(* CODESYS project EcoWatt.library
   Description: This library retrieve EcoWatt indicators from RTE.
   Author: quenorha
   Version: 1.0.0.0
   Company: WAGO_FR
   Title: EcoWatt
   Placeholder: EcoWatt
   DocFormat: reStructuredText
   DefaultNamespace: EcoWatt

Project tree, tasks and I/O mapping:
  libraries: WagoSysVersion, 1.0.0.0 (WAGO); WagoAppJSON, 1.1.0.25 (WAGO); WagoAppString, 1.6.3.4 (WAGO); WagoAppTime, 1.7.3.5 (WAGO); WagoAppHTTP, 1.7.3.4 (WAGO)
  10 Documentation/
    function block Help [ST]
  20 Program Organization Units/
    function block FbEcoWatt [ST]
  80 Data Types/
    data type typDayEcoWatt
  30 Visualizations/
    visualisation EcoWattDay
    visualisation EcoWattHour
    visualisation EcoWattVisu
  90 Internal/
    function block FbEcoWattJSON_Handler [ST]: JSON_KeyDetected, JSON_ValueDetected
    function FuCustomFormatToDT [ST]
    function FuDTToCustomFormat [ST]
  global variables VersionHistory
  Images/
    WAGO
  00000000-0000-0000-0000-000000000000|C:\Users\u044132\Downloads\old PC\Pictures\WAGO.bmp
  text list GlobalTextList
*)

// 80 Data Types/typDayEcoWatt
TYPE typDayEcoWatt :
STRUCT
		sMessage : STRING(1024);
		dtGenDate : DT;
		dtForecastDay : DT;
		bDayValue :BYTE;
		abForecast : ARRAY [0..23] OF BYTE; 
END_STRUCT
END_TYPE

// VersionHistory
(* 

**EcoWatt.library**

Description: Library for  WAGO I/O- System 

============ =========== ====================== =================
**date**     **version** **author**             **change**       
------------ ----------- ---------------------- -----------------
11.10.2022	   1.0.0.0       quenorha          First version
============ =========== ====================== =================

**Known Bugs**
   - 
   - 

**To-Do's**
   - 
   - 

*)

VAR_GLOBAL
	Info : ProjectInfo('1.0.0.0','EcoWatt.library',sLicense:='WAGO');
END_VAR

(*

11.10.2022	   1.0.0.0       quenorha          
	* [NEW] First version
	* [FIXED] ....

*)

// 90 Internal/FbEcoWattJSON_Handler
(*
	This function block uses the methods JSON_Key_Detected, JSON_ObjcectClosed and JSON_ValueDetected to import the values of
	interest to the appropriate function block.

	
*)
FUNCTION_BLOCK FbEcoWattJSON_Handler EXTENDS FbJSON_Handler
VAR_IN_OUT
	atypEcoWatt : ARRAY [0..3] OF typDayEcoWatt;
END_VAR
VAR
	parserState					: INT;	
	m							: INT;
	bDay : INT;
	bHour: INT;
END_VAR

(*

**Function**

	
**Graphical Illustration**

	.. wago.autoimage::
	
*)
METHOD JSON_KeyDetected 
VAR_INPUT
	sJSON_Object			:	STRING; // JSON object detected
END_VAR

VAR

END_VAR


IF sJSON_Object='signals' THEN	
	parserstate:=0;// jetzt kommt der Wert
ELSIF sJSON_Object='GenerationFichier' THEN	
	parserstate:=1;// jetzt kommt der Wert
ELSIF sJSON_Object='jour' THEN	
	parserstate:=2;// jetzt kommt der Wert
ELSIF sJSON_Object='dvalue' THEN	
	parserstate:=3;// jetzt kommt der Wert	
ELSIF sJSON_Object='message' THEN	
	parserstate:=4;// jetzt kommt der Wert
ELSIF sJSON_Object='values' THEN	
	parserstate:=5;// jetzt kommt der Wert
ELSIF sJSON_Object='pas' THEN	
	parserstate:=6;// jetzt kommt der Wert	
ELSIF sJSON_Object='hvalue' THEN	
	parserstate:=7;// jetzt kommt der Wert
END_IF
END_METHOD

(*

**Function**

	

**Graphical Illustration**

	.. wago.autoimage::
	
*)
METHOD JSON_ValueDetected 
VAR_INPUT
	sJSON_Value			:	STRING(JSON_MAX_STRING_SAX); // JSON value detected
END_VAR

VAR

END_VAR
{warning disable C0371}
IF __ISVALIDREF(atypEcoWatt)=FALSE THEN
	RETURN;
END_IF

CASE parserState OF
	0: bDay:=0 ;
	   bHour:=0;
	
	1:atypEcoWatt[bDay].dtGenDate:=FuCustomFormatToDT(sDateTimeString:=sJSON_Value,sCustomFormat:='AAAA-MM-JJThh:mm:SS');
	
	2:atypEcoWatt[bDay].dtForecastDay:=FuCustomFormatToDT(sDateTimeString:=sJSON_Value,sCustomFormat:='AAAA-MM-JJThh:mm:SS');
		
	3:atypEcoWatt[bDay].bDayValue:=TO_BYTE(sJSON_Value);
	
	4:atypEcoWatt[bDay].sMessage:=sJSON_Value;
		
	5://atypEcoWatt[bDay].abForecast[bHour]:=TO_BYTE(sJSON_Value);
		
	
	6:bHour:=TO_BYTE(sJSON_Value);
		
	7:atypEcoWatt[bDay].abForecast[bHour]:=TO_BYTE(sJSON_Value);
		IF bHour=23 THEN
			bDay:=bDay+1;
		END_IF

END_CASE
{warning enable C0371}
END_METHOD

END_FUNCTION_BLOCK

// 90 Internal/FuCustomFormatToDT
FUNCTION FuCustomFormatToDT : DT
(*This function returns the date/time value into a string formated with a customizable format, for example JJ/MM/AA,HH:mm:SS*)
VAR_INPUT
	sDateTimeString :  STRING ; (*Date/Time to format*)
	sCustomFormat : STRING :='JJ/MM/AA,HH:mm:SS'; (*Date/Time format to use, for example JJ/MM/AA,HH:mm:SS*)
END_VAR
VAR
	sYear : STRING(4);
	sShortYear : STRING(2);
 	sMonth :  STRING(2);
	sDay : STRING(2);
	sHour : STRING(2);
	sMinute : STRING(2);
	sSecond : STRING(2);
	sTemp:STRING;
	sTempResult : STRING;
	sSeparator : STRING(1);
	sFormat : STRING;
	i : INT;
	xAdd : BOOL;
	
	iPos : INT;
	iLength : INT;
	bSecond: BYTE;
	bMinute: BYTE;
	bHour: BYTE;
	bMonth: BYTE;
	bDay: BYTE;
	wYear: WORD;
END_VAR

IF sDateTimeString='' THEN
	FuCustomFormatToDT:=dt#1970-01-01-00:00:00;
ELSE
	iPos:=FIND(sCustomFormat,'SS');
	IF iPos=0 THEN
		iPos:=FIND(sCustomFormat,'ss');	
	END_IF
	IF iPos=0 THEN
		sSecond:='00';
	ELSE
		sSecond:=MID(sDateTimeString,2,iPos);
	END_IF
	bSecond:=STRING_TO_BYTE(sSecond);
		
	iPos:=FIND(sCustomFormat,'mm');
	IF iPos=0 THEN
		sMinute:='00';
	ELSE
		sMinute:=MID(sDateTimeString,2,iPos);
	END_IF
	bMinute:=STRING_TO_BYTE(sMinute);
		
	iPos:=FIND(sCustomFormat,'HH');
	IF iPos=0 THEN
		iPos:=FIND(sCustomFormat,'hh');	
	END_IF
	IF iPos=0 THEN
		sHour:='00';
	ELSE
		sHour:=MID(sDateTimeString,2,iPos);
	END_IF
	bHour:=STRING_TO_BYTE(sHour);
	
	
	iPos:=FIND(sCustomFormat,'MM');
	IF iPos=0 THEN
		sMonth:='00';
	ELSE
		sMonth:=MID(sDateTimeString,2,iPos);
	END_IF
	bMonth:=STRING_TO_BYTE(sMonth);
		
	iPos:=FIND(sCustomFormat,'JJ');
	IF iPos=0 THEN
		iPos:=FIND(sCustomFormat,'jj');	
	END_IF
	IF iPos=0 THEN
		sDay:='00';
	ELSE
		sDay:=MID(sDateTimeString,2,iPos);
	END_IF
	bDay:=STRING_TO_BYTE(sDay);	
	
	iPos:=FIND(sCustomFormat,'AAAA');
	iLength:=4;
	IF iPos=0 THEN
		iPos:=FIND(sCustomFormat,'aaaa');
		iLength:=4;	
	END_IF
	IF iPos=0 THEN
		iPos:=FIND(sCustomFormat,'AA');
		iLength:=2;	
	END_IF
	IF iPos=0 THEN
		iPos:=FIND(sDateTimeString,'aa');
		iLength:=2;	
	END_IF
	IF iPos=0 THEN
		sYear:='00';
	ELSE
		sYear:=MID(sDateTimeString,iLength,iPos);
	END_IF
	IF iLength=2 THEN
		wYear:=STRING_TO_WORD(sYear);
		wYear:=wYear+2000;		
	ELSE	
		wYear:=STRING_TO_WORD(sYear);	
	END_IF
	
	FuCustomFormatToDT:=FuFormatToDT(bDay,bMonth,TO_INT(wYear),bHour,bMinute,bSecond);	
END_IF

END_FUNCTION

// 10 Documentation/Help
(*

.. note::  Note

**Bibliothèque EcoWatt**
///Cette bibliothèque permet de Récupérer les informations du signal EcoWatt fournies par RTE. 
///Créer un compte sur https://data.rte-france.com/catalog/-/api/consumption/Ecowatt/v4.0
///S'abonner à l'API EcoWatt. 
///Dans "mes applications", Cliquer sur Copier en base 64 pour récupérer l'identifiant. 
///Le renseigner au niveau de sBase64Code.
///Lorsque xUpdate est activé, la requête de récupération du jeton est effectué, puis la requête de récupération des données. 
///xUpdate retombe à FALSE lorsque la requête est effectuée ou si il y a une erreur.

///Les valeurs numériques retournées correspondent aux niveaux suivant : 
/// - 1) Vert : La consommation est normale
/// - 2) Orange : le système électrique est tendu : "écogestes" bienvenus.
/// - 3) Rouge : le système électrique est très tendu, coupures inévitables si la consommation n'est pas réduite. 
///bCurrentEcoWattValue et bextEcoWattValue fournissent la valeur EcoWatt de l'heure en cours et de l'heure suivante. 
///Attention à faire en sorte de rafraichir les données périodiquement en activant xUpdate. 
///L'API ne peut être appelée que toutes les 15 minutes. Au delà de ce quota, le code HTTP 429 sera renvoyé.

	
.. figure:: ../../images/WAGO.bmp
	:align: center
	:alt: descriptif de l'image
	
*)
FUNCTION_BLOCK Help

END_FUNCTION_BLOCK

// 20 Program Organization Units/FbEcoWatt

///Cette bibliothèque permet de Récupérer les informations du signal EcoWatt fournies par RTE. 
///Créer un compte sur https://data.rte-france.com/catalog/-/api/consumption/Ecowatt/v4.0
///S'abonner à l'API EcoWatt. 
///Dans "mes applications", Cliquer sur Copier en base 64 pour récupérer l'identifiant. 
///Le renseigner au niveau de sBase64Code.
///Lorsque xUpdate est activé, la requête de récupération du jeton est effectué, puis la requête de récupération des données. 
///xUpdate retombe à FALSE lorsque la requête est effectuée ou si il y a une erreur.

///Les valeurs numériques retournées correspondent aux niveaux suivant : 
/// - 1) Vert : La consommation est normale
/// - 2) Orange : le système électrique est tendu : "écogestes" bienvenus.
/// - 3) Rouge : le système électrique est très tendu, coupures inévitables si la consommation n'est pas réduite. 
///bCurrentEcoWattValue et bextEcoWattValue fournissent la valeur EcoWatt de l'heure en cours et de l'heure suivante. 
///Attention à faire en sorte de rafraichir les données périodiquement en activant xUpdate. 
///L'API ne peut être appelée que toutes les 15 minutes. Au delà de ce quota, le code HTTP 429 sera renvoyé.

FUNCTION_BLOCK FbEcoWatt
VAR_INPUT
	sBase64Code : STRING(255); //Identifiant API RTE au format base 64.
END_VAR
VAR_IN_OUT 
	xUpdate: BOOL;				// Rafraichit les données - retombe automatiquement. 
END_VAR
VAR_OUTPUT
	atypEcoWatt : ARRAY [0..3] OF typDayEcoWatt; // Données EcoWatt aujourd'hui, et jusqu'à J+3
	bCurrentEcoWattValue : BYTE;   // Indicateur EcoWatt heure en cours 
	bNextEcoWattValue : BYTE; // Indicateur EcoWatt heure suivante
	xError : BOOL;
	sErrorDesc: STRING;
END_VAR
VAR
	oFbHTTPs_Get_Token: WagoAppHTTP.FbHTTPs_Get;
	xTriggerToken: BOOL;
	sBuffer : STRING(3000);
	sExempleData : STRING(3000):='{"signals": [{"GenerationFichier": "2022-10-10T07:36:25+02:00","jour": "2022-10-10T00:00:00+02:00","dvalue": 1,"message": "Situation normale ","values": [{"pas": 0,"hvalue": 1},{"pas": 1,"hvalue": 1},{"pas": 2,"hvalue": 1},{"pas": 3,"hvalue": 1},{"pas": 4,"hvalue": 1},{"pas": 5,"hvalue": 1},{"pas": 6,"hvalue": 1},{"pas": 7,"hvalue": 1},{"pas": 8,"hvalue": 1},{"pas": 9,"hvalue": 1},{"pas": 10,"hvalue": 1},{"pas": 11,"hvalue": 1},{"pas": 12,"hvalue": 1},{"pas": 13,"hvalue": 1},{"pas": 14,"hvalue": 1},{"pas": 15,"hvalue": 1},{"pas": 16,"hvalue": 1},{"pas": 17,"hvalue": 1},{"pas": 18,"hvalue": 1},{"pas": 19,"hvalue": 1},{"pas": 20,"hvalue": 1},{"pas": 21,"hvalue": 1},{"pas": 22,"hvalue": 1},{"pas": 23,"hvalue": 1}]},{"GenerationFichier": "2022-10-11T07:36:25+02:00","jour": "2022-10-11T00:00:00+02:00","dvalue": 3,"message": "Coupures d$'électricité programmées","values": [{"pas": 0,"hvalue": 1},{"pas": 1,"hvalue": 1},{"pas": 2,"hvalue": 1},{"pas": 3,"hvalue": 1},{"pas": 4,"hvalue": 1},{"pas": 5,"hvalue": 2},{"pas": 6,"hvalue": 2},{"pas": 7,"hvalue": 3},{"pas": 8,"hvalue": 3},{"pas": 9,"hvalue": 3},{"pas": 10,"hvalue": 3},{"pas": 11,"hvalue": 3},{"pas": 12,"hvalue": 3},{"pas": 13,"hvalue": 2},{"pas": 14,"hvalue": 2},{"pas": 15,"hvalue": 2},{"pas": 16,"hvalue": 2},{"pas": 17,"hvalue": 3},{"pas": 18,"hvalue": 3},{"pas": 19,"hvalue": 3},{"pas": 20,"hvalue": 2},{"pas": 21,"hvalue": 2},{"pas": 22,"hvalue": 2},{"pas": 23,"hvalue": 2}]},{"GenerationFichier": "2022-10-12T07:36:25+02:00","jour": "2022-10-12T00:00:00+02:00","dvalue": 2,"message": "Risque de coupures d$'électricité","values": [{"pas": 0,"hvalue": 1},{"pas": 1,"hvalue": 1},{"pas": 2,"hvalue": 1},{"pas": 3,"hvalue": 1},{"pas": 4,"hvalue": 1},{"pas": 5,"hvalue": 1},{"pas": 6,"hvalue": 1},{"pas": 7,"hvalue": 2},{"pas": 8,"hvalue": 2},{"pas": 9,"hvalue": 2},{"pas": 10,"hvalue": 2},{"pas": 11,"hvalue": 2},{"pas": 12,"hvalue": 1},{"pas": 13,"hvalue": 1},{"pas": 14,"hvalue": 1},{"pas": 15,"hvalue": 1},{"pas": 16,"hvalue": 1},{"pas": 17,"hvalue": 2},{"pas": 18,"hvalue": 2},{"pas": 19,"hvalue": 1},{"pas": 20,"hvalue": 1},{"pas": 21,"hvalue": 1},{"pas": 22,"hvalue": 1},{"pas": 23,"hvalue": 1}]},{"GenerationFichier": "2022-06-03T07:36:25+02:00","jour": "2022-10-13T00:00:00+02:00","dvalue": 3,"message": "Coupures d$'électricité en cours","values": [{"pas": 0,"hvalue": 1},{"pas": 1,"hvalue": 1},{"pas": 2,"hvalue": 1},{"pas": 3,"hvalue": 1},{"pas": 4,"hvalue": 1},{"pas": 5,"hvalue": 1},{"pas": 6,"hvalue": 1},{"pas": 7,"hvalue": 3},{"pas": 8,"hvalue": 3},{"pas": 9,"hvalue": 1},{"pas": 10,"hvalue": 1},{"pas": 11,"hvalue": 1},{"pas": 12,"hvalue": 1},{"pas": 13,"hvalue": 1},{"pas": 14,"hvalue": 3},{"pas": 15,"hvalue": 3},{"pas": 16,"hvalue": 3},{"pas": 17,"hvalue": 3},{"pas": 18,"hvalue": 3},{"pas": 19,"hvalue": 3},{"pas": 20,"hvalue": 3},{"pas": 21,"hvalue": 2},{"pas": 22,"hvalue": 2},{"pas": 23,"hvalue": 2}]}]}';
	sToken: WagoAppString.maxString;
	oFbHTTPs_Get_EcoWattSignal: WagoAppHTTP.FbHTTPs_Get;
	xTriggerSignal: BOOL;
	iStep: INT;

	oFbHTTPs_Get: WagoAppHTTP.FbHTTPs_Get;
	sURI: STRING(1023);
	sHeader: STRING(1023);
	xTrigger: BOOL;
	sEcoWattResult: STRING(1000);
	
	
	
	oFbJSON_Sax_Parser: FbJSON_Sax_Parser(oFbEcoWattJSON_Handler);
	xTriggerJSONParser: BOOL;
	oFbEcoWattJSON_Handler: FbEcoWattJSON_Handler;
	
	
	dtActualDateAndTime: DATE_AND_TIME;
	dtUpdate : DATE_AND_TIME;
	LocalTimeComponents: WagoTypes.typWagoTimeComponents;
	LocalTimeComponentsToday: WagoTypes.typWagoTimeComponents;
	
	xDemo : BOOL:=FALSE;
	oTon1m : TON;
		oStatus: WagoAppHTTP.WagoSysErrorBase.FbResult;
END_VAR


	CASE iStep OF 
		
		0 : IF xUpdate THEN
				iStep:=iStep+1;
				sURI:='https://digital.iservices.rte-france.com/token/oauth/';
				sHeader:=CONCAT('Authorization: Basic ',sBase64Code);
				xTrigger:=TRUE;
				xError:=FALSE;
				sErrorDesc:='';
				
			END_IF	
			
		1 : IF NOT xTrigger THEN
				IF oFbHTTPs_Get.xError THEN
					iStep:=99;
					oStatus:=oFbHTTPs_Get.oStatus;
				ELSE
					sToken := StrExtractSub(sBuffer,SIZEOF(sBuffer), 23, 54) ; 
					sURI:='https://digital.iservices.rte-france.com/open_api/ecowatt/v4/signals';
					sHeader:=CONCAT('Authorization: Bearer ',sToken);
					xTrigger:=TRUE;
					iStep:=iStep+1;
				END_IF
			END_IF
			
		2:	IF NOT xTrigger THEN
				IF oFbHTTPs_Get.xError THEN
					iStep:=99;
					oStatus:=oFbHTTPs_Get.oStatus;
				ELSE
					IF xDemo THEN
						sBuffer:=sExempleData;
					END_IF
					//sEcoWattResult := sBuffer;
					sURI:='https://digital.iservices.rte-france.com/open_api/ecowatt/v4/signals';
					xTriggerJSONParser:=TRUE;
					iStep:=iStep+1;
					
				END_IF
			END_IF
			
		3 : IF NOT xTriggerJSONParser THEN
				IF oFbJSON_Sax_Parser.xError THEN
					iStep:=99;
					oStatus:=oFbJSON_Sax_Parser.oStatus;
				ELSE
					iStep:=0;
					xUpdate:=FALSE;
					dtUpdate:=WagoAppTime.FuGetLocalDateAndTime();
				END_IF
			END_IF
				
	
	
		99 : sErrorDesc:= oStatus.GetDescription();
			 iStep:=0;
			 xUpdate:=FALSE;
			 xError:=TRUE;
			
	END_CASE
	
	oTon1m(IN:=NOT oTon1m.Q, PT:=T#1M);
	
	IF oTon1m.Q THEN //check every minute
		dtActualDateAndTime := WagoAppTime.FuGetLocalDateAndTime();
	
		LocalTimeComponents:=FuConvertStampToLocalTimeComponents(dtStamp:=dtActualDateAndTime );
		LocalTimeComponentsToday:=FuConvertStampToLocalTimeComponents(dtStamp:=atypEcoWatt[0].dtForecastDay );
		
		IF LocalTimeComponents.uiDay=LocalTimeComponentsToday.uiDay AND LocalTimeComponents.uiMonth=LocalTimeComponentsToday.uiMonth AND LocalTimeComponents.uiYear=LocalTimeComponentsToday.uiYear  THEN
			bCurrentEcoWattValue:=atypEcoWatt[0].abForecast[LocalTimeComponents.uiHour];
			IF LocalTimeComponents.uiHour=23 THEN
				bNextEcoWattValue:=atypEcoWatt[0].abForecast[LocalTimeComponents.uiHour];
			ELSE	
				bNextEcoWattValue:=atypEcoWatt[1].abForecast[0];
			END_IF
			
		END_IF
	END_IF
	
	
	oFbHTTPs_Get(
	sURI:=sURI , 
	sUser:=,
	sPassword:= , 
	sHeader:=sHeader,
	eAuthentication:=0 , 
	pRxBuffer:=ADR(sBuffer) , 
	udiRxBufferSize:=SIZEOF(sBuffer) , 
	tTimeout:=T#5S , 
	typSSL_Options:= , 
	xTrigger:=xTrigger, 
	xBusy=> , 
	xError=> , 
	oStatus=>oStatus , 
	udiRxNBytes=> );
		
	oFbEcoWattJSON_Handler(atypEcoWatt:=atypEcoWatt );

	oFbJSON_Sax_Parser(
	pData:=ADR(sBuffer) , 
	udiSizeData:=SIZEOF(sBuffer) , 
	sFileName:= , 
	xTrigger:=xTriggerJSONParser , 
	oStatus=> , 
	xDone=> , 
	xError=> , 
	udiValueCount=> , 
	iChunksCompleted=> );

END_FUNCTION_BLOCK

// 90 Internal/FuDTToCustomFormat
FUNCTION FuDTToCustomFormat : STRING
(*This function returns the date/time value into a string formated with a customizable format, for example JJ/MM/AA,HH:mm:SS*)
VAR_INPUT
	dtDateTime : DT; (*Date/Time to format*)
	sCustomFormat : STRING :='JJ/MM/AA,HH:mm:SS'; (*Date/Time format to use, for example JJ/MM/AA,HH:mm:SS*)
END_VAR
VAR
	sYear : STRING(4);
	sShortYear : STRING(2);
 	sMonth :  STRING(2);
	sDay : STRING(2);
	sHour : STRING(2);
	sMinute : STRING(2);
	sSecond : STRING(2);
	sTemp:STRING;
	sTempResult : STRING;
	sSeparator : STRING(1);
	sFormat : STRING;
	i : INT;
	xAdd : BOOL;
END_VAR

IF dtDateTime=dt#1970-01-01-00:00:00 THEN
	FuDTToCustomFormat:='-';
ELSE
	
	sYear := MID(DT_TO_STRING(dtDateTime),4,4);
	sShortYear := MID(DT_TO_STRING(dtDateTime),2,6);
	sMonth := MID(DT_TO_STRING(dtDateTime),2,9);
	sDay := MID(DT_TO_STRING(dtDateTime),2,12);
	sHour := MID(DT_TO_STRING(dtDateTime),2,15);
	sMinute := MID(DT_TO_STRING(dtDateTime),2,18);
	sSecond := MID(DT_TO_STRING(dtDateTime),2,21);
	
	IF LEN(sShortYear)<2 THEN
	sShortYear:=CONCAT('0',sShortYear);
	END_IF
	IF LEN(sMonth)<2 THEN
	sMonth:=CONCAT('0',sMonth);
	END_IF
	IF LEN(sDay)<2 THEN
	sDay:=CONCAT('0',sDay);
	END_IF
	IF LEN(sHour)<2 THEN
	sHour:=CONCAT('0',sHour);
	END_IF
	IF LEN(sMinute)<2 THEN
	sMinute:=CONCAT('0',sMinute);
	END_IF
	IF LEN(sSecond)<2 THEN
	sSecond:=CONCAT('0',sSecond);
	END_IF
	
	sTemp:='';
	sTempResult:='';
	
	IF sCustomFormat='' THEN
		sFormat:='JJ/MM/AA,HH:mm:SS';
	ELSE
		sFormat:=sCustomFormat;
	END_IF
	
	FOR i:=1 TO LEN(sFormat)+1 DO
	
				IF sTemp<>'' THEN (*Vérification si première itération*)
					IF MID(sFormat,1,i) = MID(sTemp,1,1)  THEN (*Vérification si Changement lettre*)
					sTemp:=CONCAT(sTemp,MID(sFormat,1,i));
					ELSE
					xAdd:=TRUE;
					END_IF
				ELSE	(*Première itération*)
					IF  MID(sFormat,1,i) <> 'J' AND MID(sFormat,1,i) <> 'j' AND MID(sFormat,1,i) <> 'M' AND MID(sFormat,1,i) <> 'A' AND MID(sFormat,1,i) <> 'a'  AND MID(sFormat,1,i) <> 'H' AND MID(sFormat,1,i) <> 'h' AND MID(sFormat,1,i) <> 'm' AND MID(sFormat,1,i) <> 'S' AND MID(sFormat,1,i) <> 's' THEN
					xAdd :=TRUE;
					ELSE
					sTemp:=CONCAT(sTemp,MID(sFormat,1,i));
					END_IF
				END_IF
	
		IF xAdd THEN
	
			IF sTemp='JJ' OR sTemp='jj' THEN
				sTempResult:=CONCAT(sTempResult,sDay);
			ELSIF sTemp='MM' THEN
				sTempResult:=CONCAT(sTempResult,sMonth);
			ELSIF sTemp='AA' OR sTemp='aa'  THEN
				sTempResult:=CONCAT(sTempResult,sShortYear);
			ELSIF sTemp='AAAA' OR sTemp='aaaa' THEN
				sTempResult:=CONCAT(sTempResult,sYear);
			ELSIF sTemp='HH' OR  sTemp='hh'  THEN
				sTempResult:=CONCAT(sTempResult,sHour);
			ELSIF sTemp='mm' THEN
				sTempResult:=CONCAT(sTempResult,sMinute);
			ELSIF sTemp='SS' OR sTemp='ss' THEN
				sTempResult:=CONCAT(sTempResult,sSecond);
			END_IF
	
			IF  MID(sFormat,1,i) <> 'J' AND MID(sFormat,1,i) <> 'j' AND MID(sFormat,1,i) <> 'M' AND MID(sFormat,1,i) <> 'A' AND MID(sFormat,1,i) <> 'a'  AND MID(sFormat,1,i) <> 'H' AND MID(sFormat,1,i) <> 'h' AND MID(sFormat,1,i) <> 'm' AND MID(sFormat,1,i) <> 'S' AND MID(sFormat,1,i) <> 's' THEN
					sSeparator:=MID(sFormat,1,i);
					sTempResult:=CONCAT(sTempResult,sSeparator);
					sTemp:='';
			ELSE
					sTemp:=MID(sFormat,1,i);
			END_IF
	
	
		xAdd:=FALSE;
		END_IF
	
	
	END_FOR
	
	FuDTtoCustomFormat:=sTempResult;
END_IF

END_FUNCTION

// 30 Visualizations/EcoWattDay
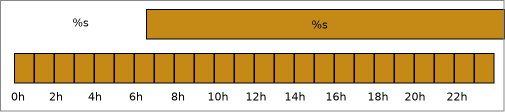
VISUALIZATION EcoWattDay  // 505x112
VAR_INPUT
	typDayEcoWatt : typDayEcoWatt;
END_VAR
    Frame (146,9 359x30)
        shows EcoWattHour(bValue := typDayEcoWatt.bDayValue)
    Frame (14,53 20x30)
        shows EcoWattHour(bValue := typDayEcoWatt.abForecast[0])
    Frame (34,53 20x30)
        shows EcoWattHour(bValue := typDayEcoWatt.abForecast[1])
    Frame (54,53 20x30)
        shows EcoWattHour(bValue := typDayEcoWatt.abForecast[2])
    Frame (74,53 20x30)
        shows EcoWattHour(bValue := typDayEcoWatt.abForecast[3])
    Frame (94,53 20x30)
        shows EcoWattHour(bValue := typDayEcoWatt.abForecast[4])
    Frame (114,53 20x30)
        shows EcoWattHour(bValue := typDayEcoWatt.abForecast[5])
    Frame (134,53 20x30)
        shows EcoWattHour(bValue := typDayEcoWatt.abForecast[6])
    Frame (154,53 20x30)
        shows EcoWattHour(bValue := typDayEcoWatt.abForecast[7])
    Frame (174,53 20x30)
        shows EcoWattHour(bValue := typDayEcoWatt.abForecast[8])
    Frame (194,53 20x30)
        shows EcoWattHour(bValue := typDayEcoWatt.abForecast[9])
    Frame (214,53 20x30)
        shows EcoWattHour(bValue := typDayEcoWatt.abForecast[10])
    Frame (234,53 20x30)
        shows EcoWattHour(bValue := typDayEcoWatt.abForecast[11])
    Frame (254,53 20x30)
        shows EcoWattHour(bValue := typDayEcoWatt.abForecast[12])
    Frame (274,53 20x30)
        shows EcoWattHour(bValue := typDayEcoWatt.abForecast[13])
    Frame (294,53 20x30)
        shows EcoWattHour(bValue := typDayEcoWatt.abForecast[14])
    Frame (314,53 20x30)
        shows EcoWattHour(bValue := typDayEcoWatt.abForecast[15])
    Frame (334,53 20x30)
        shows EcoWattHour(bValue := typDayEcoWatt.abForecast[16])
    Frame (354,53 20x30)
        shows EcoWattHour(bValue := typDayEcoWatt.abForecast[17])
    Frame (374,53 20x30)
        shows EcoWattHour(bValue := typDayEcoWatt.abForecast[18])
    Frame (394,53 20x30)
        shows EcoWattHour(bValue := typDayEcoWatt.abForecast[19])
    Frame (414,53 20x30)
        shows EcoWattHour(bValue := typDayEcoWatt.abForecast[20])
    Frame (434,53 20x30)
        shows EcoWattHour(bValue := typDayEcoWatt.abForecast[21])
    Frame (454,53 20x30)
        shows EcoWattHour(bValue := typDayEcoWatt.abForecast[22])
    Frame (474,53 20x30)
        shows EcoWattHour(bValue := typDayEcoWatt.abForecast[23])
    Rectangle (161,10 317x30), "%s", text variable: typDayEcoWatt.sMessage
    Rectangle (25,8 111x30), "%s", text variable: FuDTToCustomFormat(dtDateTime:=typDayEcoWatt.dtForecastDay , sCustomFormat:='JJ-MM-AAAA')
    Label (5,82 26x30), "0h"
    Label (43,82 26x30), "2h"
    Label (82,82 26x30), "4h"
    Label (123,82 26x30), "6h"
    Label (165,82 26x30), "8h"
    Label (205,82 26x30), "10h"
    Label (243,82 26x30), "12h"
    Label (282,82 26x30), "14h"
    Label (323,82 26x30), "16h"
    Label (365,82 26x30), "18h"
    Label (402,82 26x30), "20h"
    Label (444,82 26x30), "22h"
END_VISUALIZATION

// 30 Visualizations/EcoWattHour
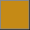
VISUALIZATION EcoWattHour  // 30x30
VAR_INPUT
	bValue : BYTE;
END_VAR
    Rectangle (0,0 30x30)
    Rectangle (0,0 30x30), invisible if: bValue<>3
    Rectangle (0,0 30x30), invisible if: bValue<>1
    Rectangle (0,0 30x30), invisible if: bValue<>2
END_VISUALIZATION

// 30 Visualizations/EcoWattVisu
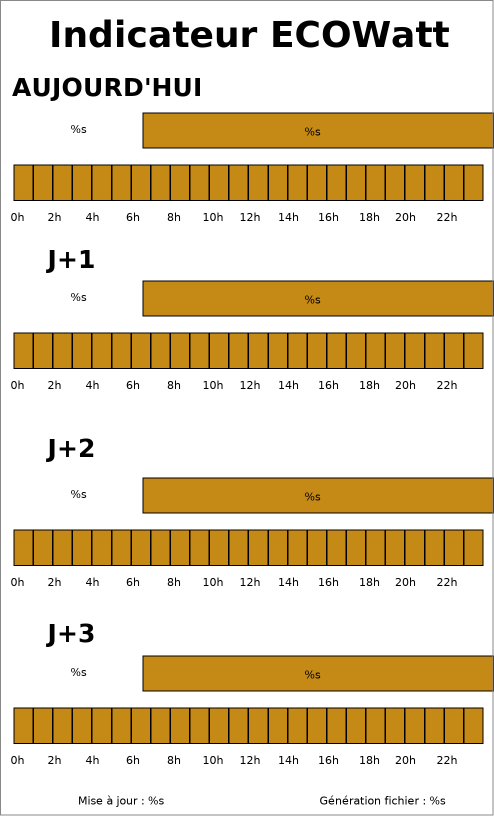
VISUALIZATION EcoWattVisu  // 494x816
VAR_IN_OUT
	FbEcoWatt : FbEcoWatt;
END_VAR
    Frame (0,102 494x133)
        shows EcoWattDay(typDayEcoWatt := FbEcoWatt.atypEcoWatt[0])
    Frame (0,270 494x133)
        shows EcoWattDay(typDayEcoWatt := FbEcoWatt.atypEcoWatt[1])
    Frame (0,467 494x133)
        shows EcoWattDay(typDayEcoWatt := FbEcoWatt.atypEcoWatt[2])
    Frame (0,645 494x133)
        shows EcoWattDay(typDayEcoWatt := FbEcoWatt.atypEcoWatt[3])
    Rectangle (276,786 213x30), "Génération fichier : %s", text variable: FuDTToCustomFormat(dtDateTime:=FbEcoWatt.atypEcoWatt[0].dtGenDate, sCustomFormat:='JJ-MM-AAAA HH:mm')
    Label (31,9 437x51), "Indicateur ECOWatt"
    Label (0,64 215x46), "AUJOURD'HUI"
    Label (0,236 143x46), "J+1"
    Label (0,425 143x46), "J+2"
    Label (0,610 143x46), "J+3"
    Rectangle (25,786 192x30), "Mise à jour : %s", text variable: FuDTToCustomFormat(dtDateTime:=FbEcoWatt.dtUpdate, sCustomFormat:='JJ-MM-AAAA HH:mm')
END_VISUALIZATION
